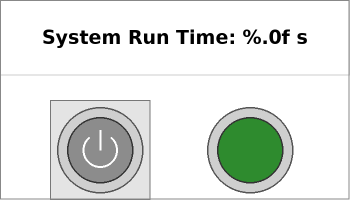
VISUALIZATION VISU_Start  // 350x200
    PowerSwitch (50,100 100x100), variable: GVL.systemRun, behaviour: TOGGLE, style: Switch-PowerSwitch-Gray
    Lamp1 (200,100 100x100), variable: GVL.bLampStart, style: Lamp-Lamp1-Green
    Textfield (0,0 350x75), "System Run Time: %.0f s", text variable: GVL.systemRunTime
END_VISUALIZATION

(* stored: Version 1.1.0.1
   Visu VISU_Start: Id {79993d33-6135-428f-b7bb-3dac593ddf45} *)
